Staubli VAL3: encodeJointFbk.pgx

public program encodeJointFbk()
  local num l_nRetVal
begin

end
